// TIA Portal V18 export
// export: Created 2026-06-08T17:01:58.5268088Z, ExportSetting WithDefaults, DisplayName Totally Integrated Automation Portal, DisplayVersion V18, DisplayName TIA Portal Openness, DisplayVersion V18, DisplayName TIA Portal Version Control Interface, DisplayVersion V18, DisplayName STEP 7 Professional, DisplayVersion V18, DisplayName STEP 7 Safety, DisplayVersion V18, DisplayName WinCC Professional, DisplayVersion V18
FUNCTION "M1_WIND_DOWN" : Void   // FC5, LAD
{ S7_Optimized_Access := 'TRUE' }
VERSION : 0.1
// stored: AutoNumber true, IsIECCheckEnabled false, SetENOAutomatically false, UDAEnableTagReadback false
BEGIN

REGION Network 1
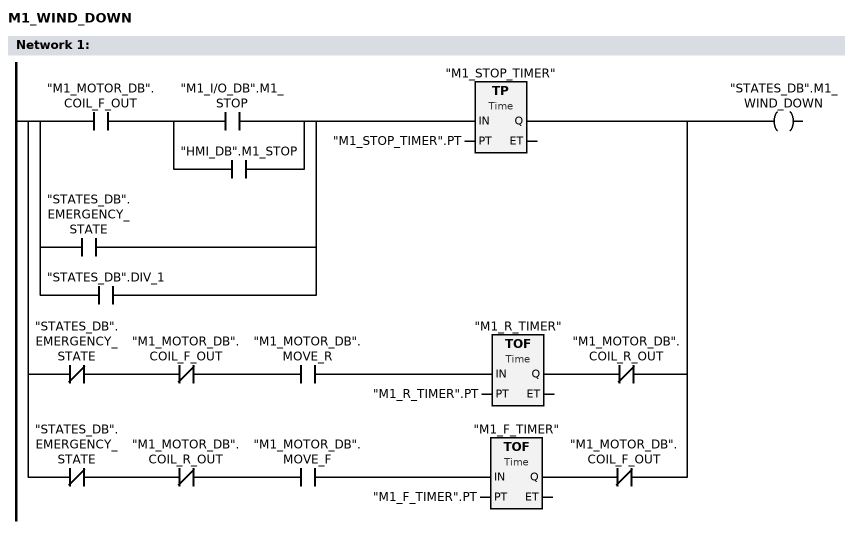
   RUNG wire#powerrail
      Contact( "M1_MOTOR_DB".COIL_F_OUT )
      wire#w1
      Contact( "M1_I/O_DB".M1_STOP )
      wire#w2
      { S7_Templates := "time_type := Time" } "M1_STOP_TIMER".TP(pt := "M1_STOP_TIMER".PT, et =>)
      wire#w3
      Coil( "STATES_DB".M1_WIND_DOWN )
   END_RUNG
   RUNG wire#w1
      Contact( "HMI_DB".M1_STOP )
   END_RUNG wire#w2
   RUNG wire#powerrail
      Contact( "STATES_DB".EMERGENCY_STATE )
   END_RUNG wire#w2
   RUNG wire#powerrail
      Contact( "STATES_DB".DIV_1 )
   END_RUNG wire#w2
   RUNG wire#powerrail
      I_Contact( "STATES_DB".EMERGENCY_STATE )
      I_Contact( "M1_MOTOR_DB".COIL_F_OUT )
      Contact( "M1_MOTOR_DB".MOVE_R )
      { S7_Templates := "time_type := Time" } "M1_R_TIMER".TOF(pt := "M1_R_TIMER".PT, et =>)
      I_Contact( "M1_MOTOR_DB".COIL_R_OUT )
   END_RUNG wire#w3
   RUNG wire#powerrail
      I_Contact( "STATES_DB".EMERGENCY_STATE )
      I_Contact( "M1_MOTOR_DB".COIL_R_OUT )
      Contact( "M1_MOTOR_DB".MOVE_F )
      { S7_Templates := "time_type := Time" } "M1_F_TIMER".TOF(pt := "M1_F_TIMER".PT, et =>)
      I_Contact( "M1_MOTOR_DB".COIL_F_OUT )
   END_RUNG wire#w3
   // the same network as SCL:
   "M1_STOP_TIMER".TP(IN := ("M1_MOTOR_DB".COIL_F_OUT AND ("M1_I/O_DB".M1_STOP OR "HMI_DB".M1_STOP)) OR "STATES_DB".EMERGENCY_STATE OR "STATES_DB".DIV_1,
                      PT := "M1_STOP_TIMER".PT);
   "M1_R_TIMER".TOF(IN := NOT "STATES_DB".EMERGENCY_STATE AND NOT "M1_MOTOR_DB".COIL_F_OUT AND "M1_MOTOR_DB".MOVE_R,
                    PT := "M1_R_TIMER".PT);
   "M1_F_TIMER".TOF(IN := NOT "STATES_DB".EMERGENCY_STATE AND NOT "M1_MOTOR_DB".COIL_R_OUT AND "M1_MOTOR_DB".MOVE_F,
                    PT := "M1_F_TIMER".PT);
   "STATES_DB".M1_WIND_DOWN := "M1_STOP_TIMER".Q OR ("M1_R_TIMER".Q AND NOT "M1_MOTOR_DB".COIL_R_OUT) OR ("M1_F_TIMER".Q AND NOT "M1_MOTOR_DB".COIL_F_OUT);
END_REGION
END_FUNCTION
